# EPICS substitutions: ek9000App/Db/EL7041.substitutions
file EL7041.template
{       pattern
        {
                TERMINAL,

        }
        {
        }
}
